// Mitsubishi GX Works2 project: 230929-001- exercicios-1   PLC: Q03UDV

// task Task_01 (event TRUE, interval 0, priority 31): POU_01

PROGRAM POU_01
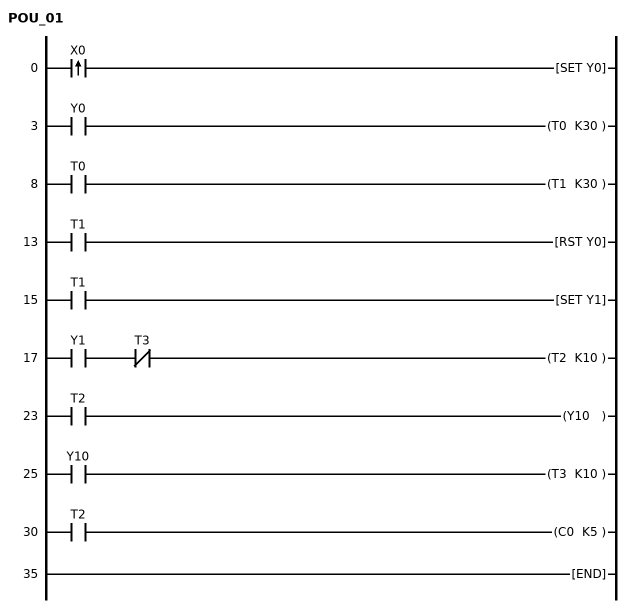
0     LDP     X0
      SET     Y0
3     LD      Y0
      OUT     T0 K30
8     LD      T0
      OUT     T1 K30
13    LD      T1
      RST     Y0
15    LD      T1
      SET     Y1
17    LD      Y1
      ANI     T3
      OUT     T2 K10
23    LD      T2
      OUT     Y10
25    LD      Y10
      OUT     T3 K10
30    LD      T2
      OUT     C0 K5
35    END
END_PROGRAM
